FUNCTION_BLOCK FB_TestFunctionBlock
VAR
	nCounter:	LINT;
END_VAR

nCounter := nCounter + 1;

END_FUNCTION_BLOCK

(* stored: Version 1.1.0.1, ProductVersion 3.1.4024.11
   POU FB_TestFunctionBlock: Id {54f8d70b-56f3-45a6-a290-b5f3e4987475}, SpecialFunc None *)
